PROGRAM MAIN
VAR
	test_input AT%I* : ARRAY [0..1] OF BOOL;
	test_output AT%Q* : ARRAY [0..1] OF BOOL;
	test_value : DINT;
	test_string: STRING(255);
END_VAR


IF test_value = 16#7FFFFFFF THEN
	test_value := 0;
END_IF

test_value := test_value + 1;

END_PROGRAM

(* stored: Version 1.1.0.1, ProductVersion 3.1.4024.12
   POU MAIN: Id {ccd35c68-4c9d-484a-a981-b7061656ed90}, SpecialFunc None *)
